// TIA Portal V17 export
// export: Created 2025-08-05T09:35:59.6415853Z, ExportSetting WithDefaults, DisplayName Totally Integrated Automation Portal, DisplayVersion V17, DisplayName TIA Portal Openness, DisplayVersion V17, DisplayName TIA Portal Version Control Interface, DisplayVersion V17, DisplayName SINAMICS Startdrive Advanced, DisplayVersion V17, DisplayName SINAMICS Startdrive G130, G150, S120, S150, SINAMICS MV, S210, DisplayVersion V17, DisplayName SINAMICS Startdrive G110M, G120, G120C, G120D, G120P, G115D, DisplayVersion V17, DisplayName STEP 7 Professional, DisplayVersion V17, DisplayName STEP 7 Safety, DisplayVersion V17, DisplayName WinCC Advanced, DisplayVersion V17
TYPE "typeFgLogEntry"
TITLE = FG log entry / FG-Log Eintrag
// FG log entry [V 01.00 | Kernel_V2] / FG-Log Eintrag [V 01.00 | Kernel_V2]
// stored: IsFailsafeCompliant false
   STRUCT
      area { ExternalAccessible := 'False'; ExternalVisible := 'False'; ExternalWritable := 'False'} : Byte;   // 16#FF Header | 16#01 Log Entry | 16#00 Empty
      pointerOrEventId { ExternalAccessible := 'False'; ExternalVisible := 'False'; ExternalWritable := 'False'} : DWord;   // Area = 16#00: Pointer auf letzten Eintrag | Area = 16#01: Event-ID / Area = 16#00: Pointer at last entry | Area = 16#01: Event ID
      opMode { ExternalAccessible := 'False'; ExternalVisible := 'False'; ExternalWritable := 'False'} : Byte;   // 16#01 Automatic | 16#02 SingleCycle | 16#04 SingleStep | 16#08 Manual | 16#10 MSO 2 | 16#20 MSO 3 | 16#40 MSO GROB
      baseFunction { ExternalAccessible := 'False'; ExternalVisible := 'False'; ExternalWritable := 'False'} : Byte;   // 16#00 Reset | 16#01 Stop is active | 16#02 Start is active | 16#03 Start is stopped | 16#04 HomePos active | 16#05 HomePos is stopped | 16#10 in HomePos | 16#20 Stop at cycle active
      cycleType { ExternalAccessible := 'False'; ExternalVisible := 'False'; ExternalWritable := 'False'} : Byte;   // 16#01 Empying Mode | 16#02 Dry Run | 16#04 WarmUp | 16#08 UserDef 1 | 16#10 UserDef 2
      groupMode { ExternalAccessible := 'False'; ExternalVisible := 'False'; ExternalWritable := 'False'} : Byte;   // 16#01 Group active | 16#02 Group in Interlinked Mode | 16#04 Interlock Bypass Mode
      actJobNum { ExternalAccessible := 'False'; ExternalVisible := 'False'; ExternalWritable := 'False'} : Int;   // Aktive Auftragsnummer / Active job number
      sequStepNum { ExternalAccessible := 'False'; ExternalVisible := 'False'; ExternalWritable := 'False'} : Int;   // Ablauf Schrittnummer / Sequence step number
      timeStamp { ExternalAccessible := 'False'; ExternalVisible := 'False'; ExternalWritable := 'False'} : Date_And_Time;   // Zeitstempel / Time stamp
   END_STRUCT;
END_TYPE
